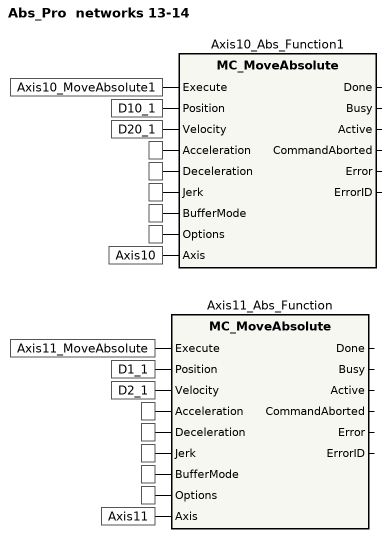
[picture p24: Abs_Pro (FBD) networks 13-14]
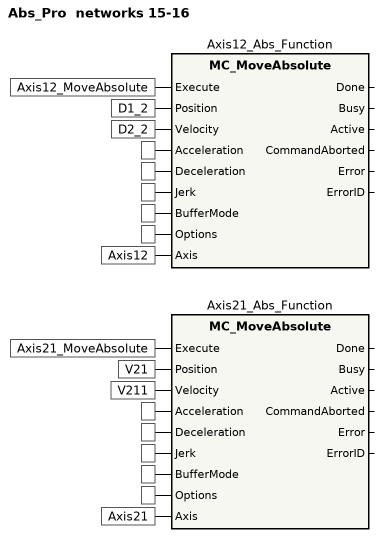
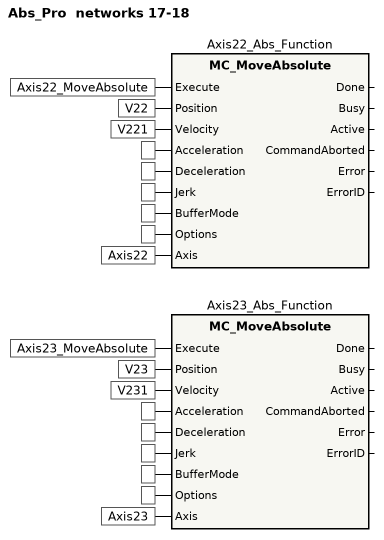
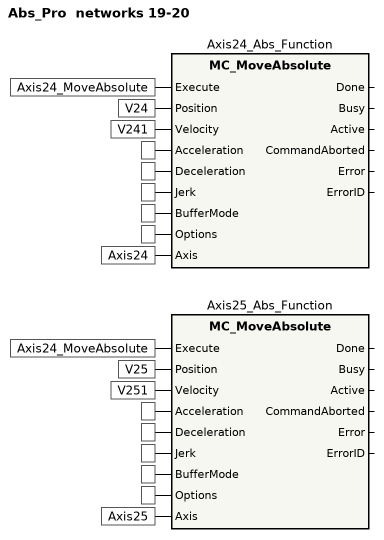
_FBD_ (* Function Block Diagram *)
NETWORK 1
	Axis1_Abs_Function:MC_MoveAbsolute(Execute: Axis1_MoveAbsolute, Position: D1, Velocity: D11, Acceleration: , Deceleration: , Jerk: , BufferMode: , Options: , Axis: Axis1)
NETWORK 2
	Axis2_Abs_Function:MC_MoveAbsolute(Execute: Axis2_MoveAbsolute, Position: D2, Velocity: D12, Acceleration: , Deceleration: , Jerk: , BufferMode: , Options: , Axis: Axis2)
NETWORK 3
	Axis3_Abs_Function:MC_MoveAbsolute(Execute: Axis3_MoveAbsolute, Position: D3, Velocity: D13, Acceleration: , Deceleration: , Jerk: , BufferMode: , Options: , Axis: Axis3)
NETWORK 4
	Axis4_Abs_Function:MC_MoveAbsolute(Execute: Axis4_MoveAbsolute, Position: D4, Velocity: D14, Acceleration: , Deceleration: , Jerk: , BufferMode: , Options: , Axis: Axis4)
NETWORK 5
	Axis4_1_Abs_Function:MC_MoveAbsolute(Execute: Axis4_1_MoveAbsolute, Position: D4, Velocity: D14_1, Acceleration: , Deceleration: , Jerk: , BufferMode: , Options: , Axis: Axis4)
NETWORK 6
	Axis5_Abs_Function:MC_MoveAbsolute(Execute: Axis5_MoveAbsolute, Position: D5, Velocity: D15, Acceleration: , Deceleration: , Jerk: , BufferMode: , Options: , Axis: Axis5)
NETWORK 7
	Axis5_1_Abs_Function:MC_MoveAbsolute(Execute: Axis5_1_MoveAbsolute, Position: D5, Velocity: D15_1, Acceleration: , Deceleration: , Jerk: , BufferMode: , Options: , Axis: Axis5)
NETWORK 8
	Axis6_Abs_Function:MC_MoveAbsolute(Execute: Axis6_MoveAbsolute, Position: D6, Velocity: D16, Acceleration: , Deceleration: , Jerk: , BufferMode: , Options: , Axis: Axis6)
NETWORK 9
	Axis7_Abs_Function:MC_MoveAbsolute(Execute: Axis7_MoveAbsolute, Position: D7, Velocity: D17, Acceleration: , Deceleration: , Jerk: , BufferMode: , Options: , Axis: Axis7)
NETWORK 10
	Axis8_Abs_Function:MC_MoveAbsolute(Execute: Axis8_MoveAbsolute, Position: D8, Velocity: D18, Acceleration: , Deceleration: , Jerk: , BufferMode: , Options: , Axis: Axis8)
NETWORK 11
	Axis9_Abs_Function:MC_MoveAbsolute(Execute: Axis9_MoveAbsolute, Position: D9, Velocity: D19, Acceleration: , Deceleration: , Jerk: , BufferMode: , Options: , Axis: Axis9)
NETWORK 12
	Axis10_Abs_Function:MC_MoveAbsolute(Execute: Axis10_MoveAbsolute, Position: D10, Velocity: D20, Acceleration: , Deceleration: , Jerk: , BufferMode: , Options: , Axis: Axis10)
NETWORK 13
	Axis10_Abs_Function1:MC_MoveAbsolute(Execute: Axis10_MoveAbsolute1, Position: D10_1, Velocity: D20_1, Acceleration: , Deceleration: , Jerk: , BufferMode: , Options: , Axis: Axis10)
NETWORK 14
	Axis11_Abs_Function:MC_MoveAbsolute(Execute: Axis11_MoveAbsolute, Position: D1_1, Velocity: D2_1, Acceleration: , Deceleration: , Jerk: , BufferMode: , Options: , Axis: Axis11)
NETWORK 15
	Axis12_Abs_Function:MC_MoveAbsolute(Execute: Axis12_MoveAbsolute, Position: D1_2, Velocity: D2_2, Acceleration: , Deceleration: , Jerk: , BufferMode: , Options: , Axis: Axis12)
NETWORK 16
	Axis21_Abs_Function:MC_MoveAbsolute(Execute: Axis21_MoveAbsolute, Position: V21, Velocity: V211, Acceleration: , Deceleration: , Jerk: , BufferMode: , Options: , Axis: Axis21)
NETWORK 17
	Axis22_Abs_Function:MC_MoveAbsolute(Execute: Axis22_MoveAbsolute, Position: V22, Velocity: V221, Acceleration: , Deceleration: , Jerk: , BufferMode: , Options: , Axis: Axis22)
NETWORK 18
	Axis23_Abs_Function:MC_MoveAbsolute(Execute: Axis23_MoveAbsolute, Position: V23, Velocity: V231, Acceleration: , Deceleration: , Jerk: , BufferMode: , Options: , Axis: Axis23)
NETWORK 19
	Axis24_Abs_Function:MC_MoveAbsolute(Execute: Axis24_MoveAbsolute, Position: V24, Velocity: V241, Acceleration: , Deceleration: , Jerk: , BufferMode: , Options: , Axis: Axis24)
NETWORK 20
	Axis25_Abs_Function:MC_MoveAbsolute(Execute: Axis24_MoveAbsolute, Position: V25, Velocity: V251, Acceleration: , Deceleration: , Jerk: , BufferMode: , Options: , Axis: Axis25)
_END_FBD_
END_PROGRAM

(* POU Other_Folder/Motion/Halt_Pro, FBD *)
PROGRAM Halt_Pro
VAR

END_VAR
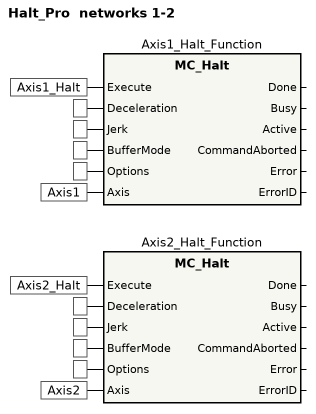
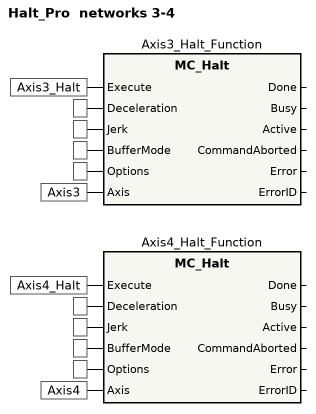
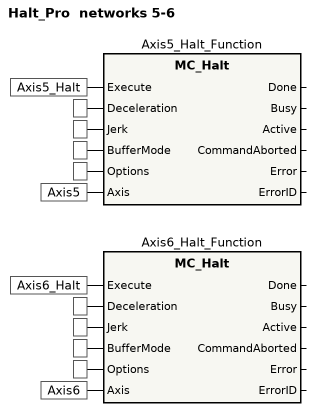
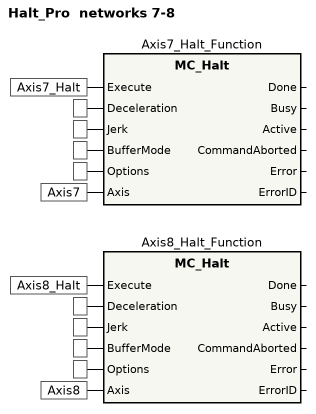
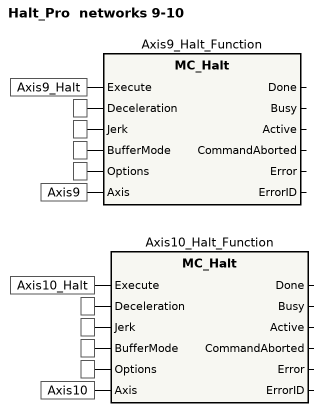
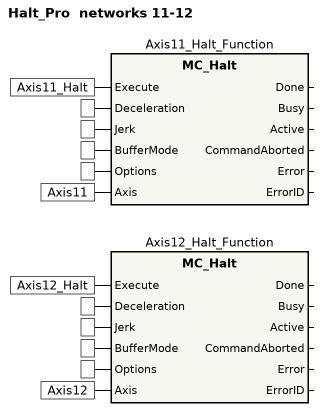
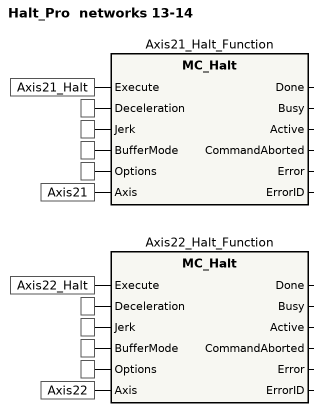
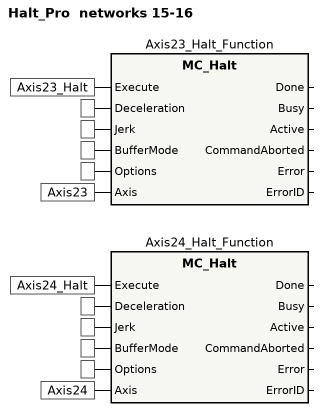
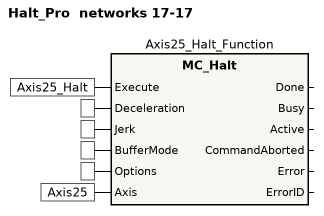
_FBD_ (* Function Block Diagram *)
NETWORK 1
	Axis1_Halt_Function:MC_Halt(Execute: Axis1_Halt, Deceleration: , Jerk: , BufferMode: , Options: , Axis: Axis1)
NETWORK 2
	Axis2_Halt_Function:MC_Halt(Execute: Axis2_Halt, Deceleration: , Jerk: , BufferMode: , Options: , Axis: Axis2)
NETWORK 3
	Axis3_Halt_Function:MC_Halt(Execute: Axis3_Halt, Deceleration: , Jerk: , BufferMode: , Options: , Axis: Axis3)
NETWORK 4
	Axis4_Halt_Function:MC_Halt(Execute: Axis4_Halt, Deceleration: , Jerk: , BufferMode: , Options: , Axis: Axis4)
NETWORK 5
	Axis5_Halt_Function:MC_Halt(Execute: Axis5_Halt, Deceleration: , Jerk: , BufferMode: , Options: , Axis: Axis5)
NETWORK 6
	Axis6_Halt_Function:MC_Halt(Execute: Axis6_Halt, Deceleration: , Jerk: , BufferMode: , Options: , Axis: Axis6)
NETWORK 7
	Axis7_Halt_Function:MC_Halt(Execute: Axis7_Halt, Deceleration: , Jerk: , BufferMode: , Options: , Axis: Axis7)
NETWORK 8
	Axis8_Halt_Function:MC_Halt(Execute: Axis8_Halt, Deceleration: , Jerk: , BufferMode: , Options: , Axis: Axis8)
NETWORK 9
	Axis9_Halt_Function:MC_Halt(Execute: Axis9_Halt, Deceleration: , Jerk: , BufferMode: , Options: , Axis: Axis9)
NETWORK 10
	Axis10_Halt_Function:MC_Halt(Execute: Axis10_Halt, Deceleration: , Jerk: , BufferMode: , Options: , Axis: Axis10)
NETWORK 11
	Axis11_Halt_Function:MC_Halt(Execute: Axis11_Halt, Deceleration: , Jerk: , BufferMode: , Options: , Axis: Axis11)
NETWORK 12
	Axis12_Halt_Function:MC_Halt(Execute: Axis12_Halt, Deceleration: , Jerk: , BufferMode: , Options: , Axis: Axis12)
NETWORK 13
	Axis21_Halt_Function:MC_Halt(Execute: Axis21_Halt, Deceleration: , Jerk: , BufferMode: , Options: , Axis: Axis21)
NETWORK 14
	Axis22_Halt_Function:MC_Halt(Execute: Axis22_Halt, Deceleration: , Jerk: , BufferMode: , Options: , Axis: Axis22)
NETWORK 15
	Axis23_Halt_Function:MC_Halt(Execute: Axis23_Halt, Deceleration: , Jerk: , BufferMode: , Options: , Axis: Axis23)
NETWORK 16
	Axis24_Halt_Function:MC_Halt(Execute: Axis24_Halt, Deceleration: , Jerk: , BufferMode: , Options: , Axis: Axis24)
NETWORK 17
	Axis25_Halt_Function:MC_Halt(Execute: Axis25_Halt, Deceleration: , Jerk: , BufferMode: , Options: , Axis: Axis25)
_END_FBD_
END_PROGRAM

(* POU Other_Folder/Speed_AxisStatus_IO/Motion_Rst, LD *)
PROGRAM Motion_Rst
VAR

END_VAR
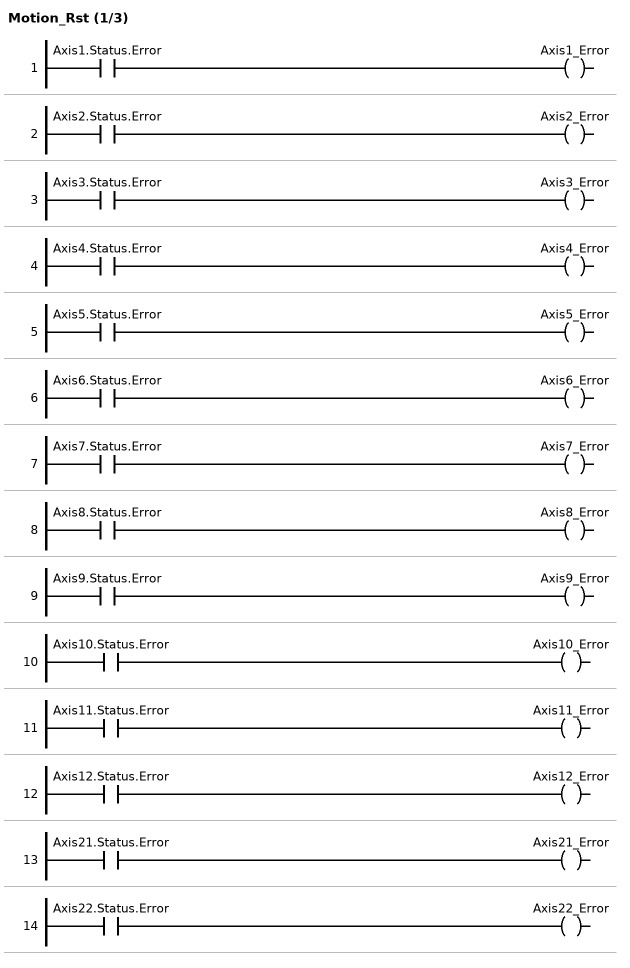
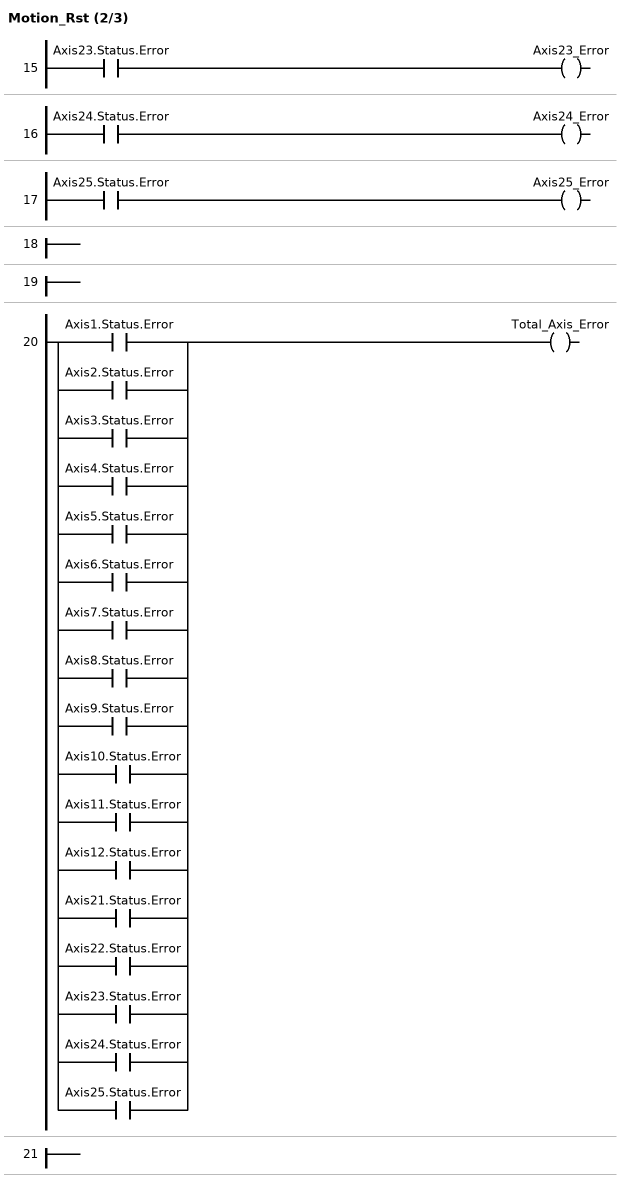
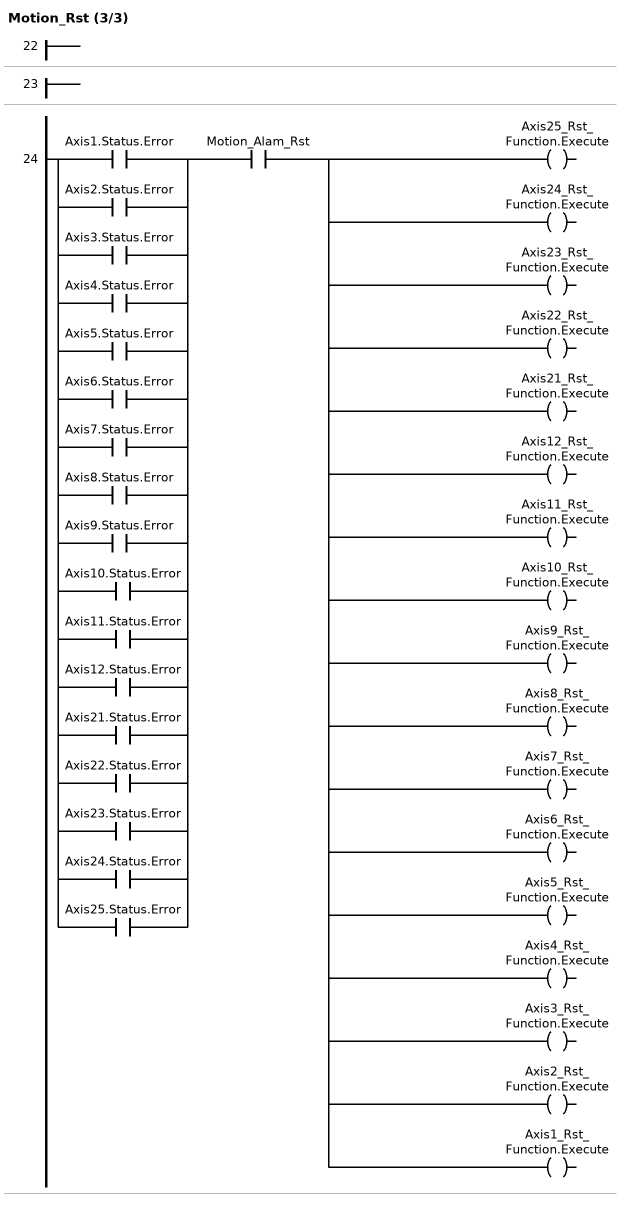
_LD_ (* Ladder Diagram *)
NETWORK 1
	[Axis1.Status.Error] --- (Axis1_Error)
NETWORK 2
	[Axis2.Status.Error] --- (Axis2_Error)
NETWORK 3
	[Axis3.Status.Error] --- (Axis3_Error)
NETWORK 4
	[Axis4.Status.Error] --- (Axis4_Error)
NETWORK 5
	[Axis5.Status.Error] --- (Axis5_Error)
NETWORK 6
	[Axis6.Status.Error] --- (Axis6_Error)
NETWORK 7
	[Axis7.Status.Error] --- (Axis7_Error)
NETWORK 8
	[Axis8.Status.Error] --- (Axis8_Error)
NETWORK 9
	[Axis9.Status.Error] --- (Axis9_Error)
NETWORK 10
	[Axis10.Status.Error] --- (Axis10_Error)
NETWORK 11
	[Axis11.Status.Error] --- (Axis11_Error)
NETWORK 12
	[Axis12.Status.Error] --- (Axis12_Error)
NETWORK 13
	[Axis21.Status.Error] --- (Axis21_Error)
NETWORK 14
	[Axis22.Status.Error] --- (Axis22_Error)
NETWORK 15
	[Axis23.Status.Error] --- (Axis23_Error)
NETWORK 16
	[Axis24.Status.Error] --- (Axis24_Error)
NETWORK 17
	[Axis25.Status.Error] --- (Axis25_Error)
NETWORK 18
	*
NETWORK 19
	*
NETWORK 20
	{ [Axis1.Status.Error] | [Axis2.Status.Error] | [Axis3.Status.Error] | [Axis4.Status.Error] | [Axis5.Status.Error] | [Axis6.Status.Error] | [Axis7.Status.Error] | [Axis8.Status.Error] | [Axis9.Status.Error] | [Axis10.Status.Error] | [Axis11.Status.Error] | [Axis12.Status.Error] | [Axis21.Status.Error] | [Axis22.Status.Error] | [Axis23.Status.Error] | [Axis24.Status.Error] | [Axis25.Status.Error] } --- (Total_Axis_Error)
NETWORK 21
	*
NETWORK 22
	*
NETWORK 23
	*
NETWORK 24
	{ [Axis1.Status.Error] | [Axis2.Status.Error] | [Axis3.Status.Error] | [Axis4.Status.Error] | [Axis5.Status.Error] | [Axis6.Status.Error] | [Axis7.Status.Error] | [Axis8.Status.Error] | [Axis9.Status.Error] | [Axis10.Status.Error] | [Axis11.Status.Error] | [Axis12.Status.Error] | [Axis21.Status.Error] | [Axis22.Status.Error] | [Axis23.Status.Error] | [Axis24.Status.Error] | [Axis25.Status.Error] } - [Motion_Alam_Rst] --- (Axis25_Rst_Function.Execute) (Axis24_Rst_Function.Execute) (Axis23_Rst_Function.Execute) (Axis22_Rst_Function.Execute) (Axis21_Rst_Function.Execute) (Axis12_Rst_Function.Execute) (Axis11_Rst_Function.Execute) (Axis10_Rst_Function.Execute) (Axis9_Rst_Function.Execute) (Axis8_Rst_Function.Execute) (Axis7_Rst_Function.Execute) (Axis6_Rst_Function.Execute) (Axis5_Rst_Function.Execute) (Axis4_Rst_Function.Execute) (Axis3_Rst_Function.Execute) (Axis2_Rst_Function.Execute) (Axis1_Rst_Function.Execute)
_END_LD_
(* the same logic as Structured Text *)
(* Network 1 *)
Axis1_Error := Axis1.Status.Error;
(* Network 2 *)
Axis2_Error := Axis2.Status.Error;
(* Network 3 *)
Axis3_Error := Axis3.Status.Error;
(* Network 4 *)
Axis4_Error := Axis4.Status.Error;
(* Network 5 *)
Axis5_Error := Axis5.Status.Error;
(* Network 6 *)
Axis6_Error := Axis6.Status.Error;
(* Network 7 *)
Axis7_Error := Axis7.Status.Error;
(* Network 8 *)
Axis8_Error := Axis8.Status.Error;
(* Network 9 *)
Axis9_Error := Axis9.Status.Error;
(* Network 10 *)
Axis10_Error := Axis10.Status.Error;
(* Network 11 *)
Axis11_Error := Axis11.Status.Error;
(* Network 12 *)
Axis12_Error := Axis12.Status.Error;
(* Network 13 *)
Axis21_Error := Axis21.Status.Error;
(* Network 14 *)
Axis22_Error := Axis22.Status.Error;
(* Network 15 *)
Axis23_Error := Axis23.Status.Error;
(* Network 16 *)
Axis24_Error := Axis24.Status.Error;
(* Network 17 *)
Axis25_Error := Axis25.Status.Error;
(* Network 18 *)
(* Network 19 *)
(* Network 20 *)
Total_Axis_Error := Axis1.Status.Error OR Axis2.Status.Error OR Axis3.Status.Error OR Axis4.Status.Error OR Axis5.Status.Error OR Axis6.Status.Error OR Axis7.Status.Error OR Axis8.Status.Error OR Axis9.Status.Error OR Axis10.Status.Error OR Axis11.Status.Error OR Axis12.Status.Error OR Axis21.Status.Error OR Axis22.Status.Error OR Axis23.Status.Error OR Axis24.Status.Error OR Axis25.Status.Error;
(* Network 21 *)
(* Network 22 *)
(* Network 23 *)
(* Network 24 *)
Axis25_Rst_Function.Execute := (Axis1.Status.Error OR Axis2.Status.Error OR Axis3.Status.Error OR Axis4.Status.Error OR Axis5.Status.Error OR Axis6.Status.Error OR Axis7.Status.Error OR Axis8.Status.Error OR Axis9.Status.Error OR Axis10.Status.Error OR Axis11.Status.Error OR Axis12.Status.Error OR Axis21.Status.Error OR Axis22.Status.Error OR Axis23.Status.Error OR Axis24.Status.Error OR Axis25.Status.Error) AND Motion_Alam_Rst;
Axis24_Rst_Function.Execute := Axis25_Rst_Function.Execute;
Axis23_Rst_Function.Execute := Axis25_Rst_Function.Execute;
Axis22_Rst_Function.Execute := Axis25_Rst_Function.Execute;
Axis21_Rst_Function.Execute := Axis25_Rst_Function.Execute;
Axis12_Rst_Function.Execute := Axis25_Rst_Function.Execute;
Axis11_Rst_Function.Execute := Axis25_Rst_Function.Execute;
Axis10_Rst_Function.Execute := Axis25_Rst_Function.Execute;
Axis9_Rst_Function.Execute := Axis25_Rst_Function.Execute;
Axis8_Rst_Function.Execute := Axis25_Rst_Function.Execute;
Axis7_Rst_Function.Execute := Axis25_Rst_Function.Execute;
Axis6_Rst_Function.Execute := Axis25_Rst_Function.Execute;
Axis5_Rst_Function.Execute := Axis25_Rst_Function.Execute;
Axis4_Rst_Function.Execute := Axis25_Rst_Function.Execute;
Axis3_Rst_Function.Execute := Axis25_Rst_Function.Execute;
Axis2_Rst_Function.Execute := Axis25_Rst_Function.Execute;
Axis1_Rst_Function.Execute := Axis25_Rst_Function.Execute;
END_PROGRAM

(* POU Other_Folder/Motion/MotionRst_Pro, FBD *)
PROGRAM MotionRst_Pro
VAR
END_VAR
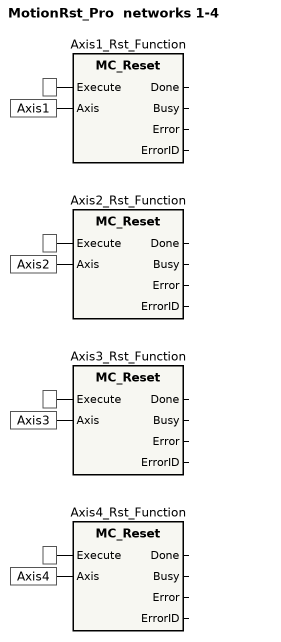
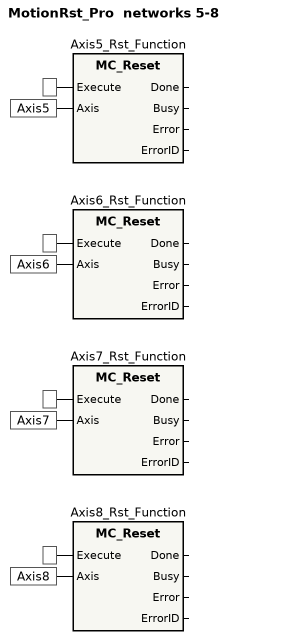
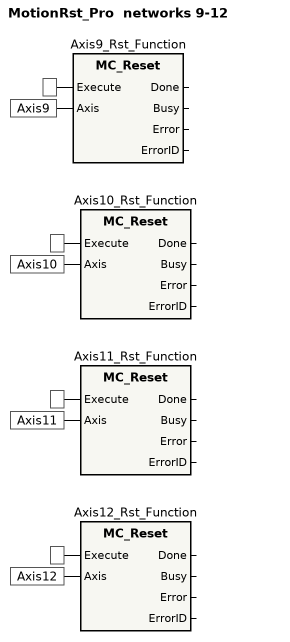
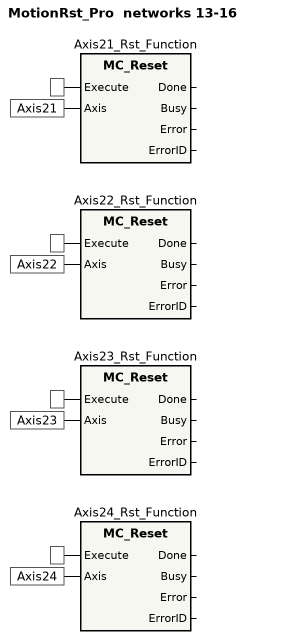
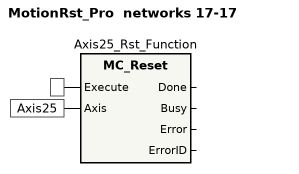
_FBD_ (* Function Block Diagram *)
NETWORK 1
	Axis1_Rst_Function:MC_Reset(Execute: , Axis: Axis1)
NETWORK 2
	Axis2_Rst_Function:MC_Reset(Execute: , Axis: Axis2)
NETWORK 3
	Axis3_Rst_Function:MC_Reset(Execute: , Axis: Axis3)
NETWORK 4
	Axis4_Rst_Function:MC_Reset(Execute: , Axis: Axis4)
NETWORK 5
	Axis5_Rst_Function:MC_Reset(Execute: , Axis: Axis5)
NETWORK 6
	Axis6_Rst_Function:MC_Reset(Execute: , Axis: Axis6)
NETWORK 7
	Axis7_Rst_Function:MC_Reset(Execute: , Axis: Axis7)
NETWORK 8
	Axis8_Rst_Function:MC_Reset(Execute: , Axis: Axis8)
NETWORK 9
	Axis9_Rst_Function:MC_Reset(Execute: , Axis: Axis9)
NETWORK 10
	Axis10_Rst_Function:MC_Reset(Execute: , Axis: Axis10)
NETWORK 11
	Axis11_Rst_Function:MC_Reset(Execute: , Axis: Axis11)
NETWORK 12
	Axis12_Rst_Function:MC_Reset(Execute: , Axis: Axis12)
NETWORK 13
	Axis21_Rst_Function:MC_Reset(Execute: , Axis: Axis21)
NETWORK 14
	Axis22_Rst_Function:MC_Reset(Execute: , Axis: Axis22)
NETWORK 15
	Axis23_Rst_Function:MC_Reset(Execute: , Axis: Axis23)
NETWORK 16
	Axis24_Rst_Function:MC_Reset(Execute: , Axis: Axis24)
NETWORK 17
	Axis25_Rst_Function:MC_Reset(Execute: , Axis: Axis25)
_END_FBD_
END_PROGRAM

(* POU Other_Folder/Motion/PTF_Pro, FBD *)
PROGRAM PTF_Pro
VAR


END_VAR
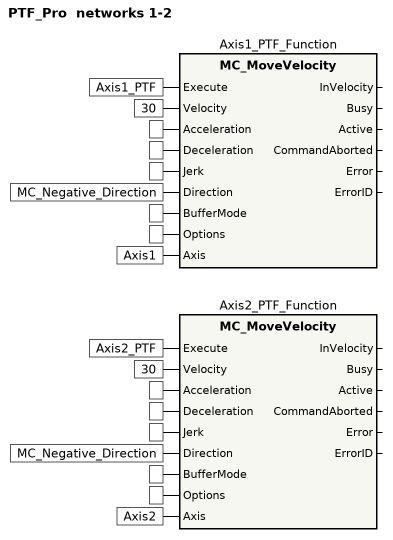
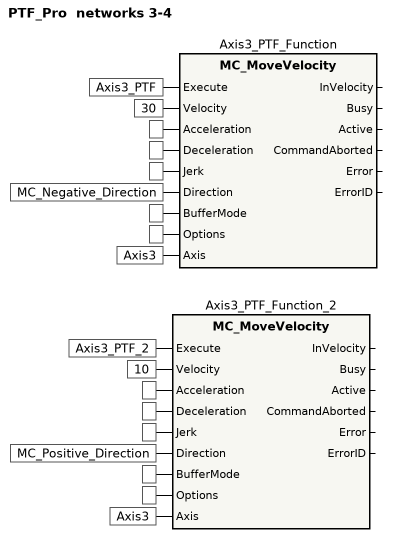
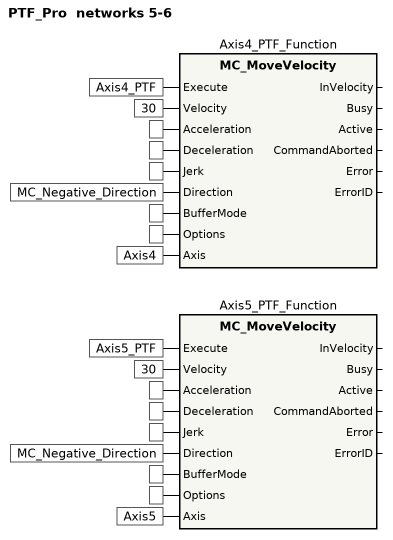
